Staubli VAL3: PickAndPlace1.dtx

bool bBool1 = true
jointRx jHome
mdesc mNomSpeed
mdesc mSlow = {accel=25, vel=25, decel=25, rmax=25, tmax=25}
num nRep
public pointRx pPointrx1[3]
  [0] = {x=498.015054, y=59.142287, z=-30.989318, rx=5.599382, ry=128.808236, rz=-7.17091, fatherId=world[0]}
  [1] = {x=445.61, y=378.050542, z=199.065349, rx=88.308613, ry=128.361913, rz=-88.673624, fatherId=world[0]}
  [2] = {x=481.810529, y=-248.36011, z=-295.450034, rx=-23.480249, ry=144.718456, rz=48.788162, fatherId=world[0]}
tool tTool1 = {fatherId=flange[0], ioLink=valve1}
